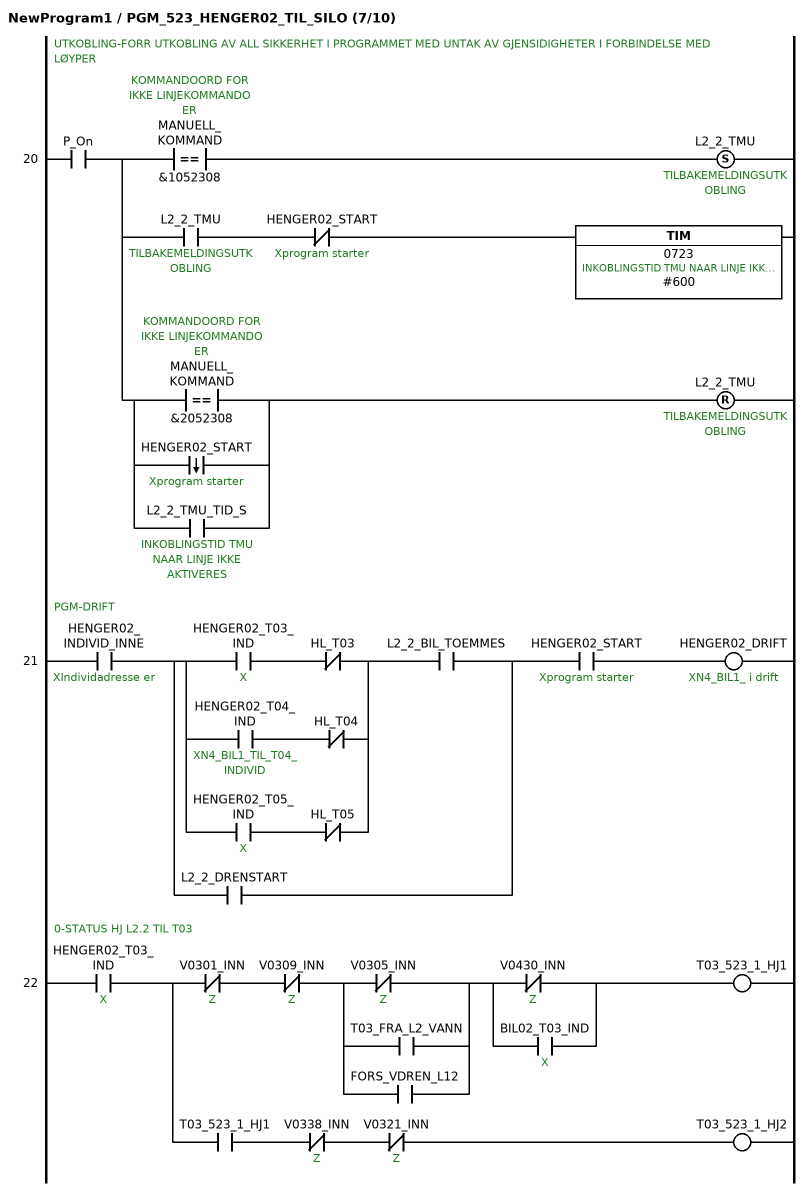
; [picture p648: NewProgram1 / PGM_523_HENGER02_TIL_SILO, rungs 20-22]
; rung 20: UTKOBLING-FORR UTKOBLING AV ALL SIKKERHET I PROGRAMMET MED UNTAK AV GJENSIDIGHETER I FORBINDELSE MED LØYPER
LD P_On
OUT TR0
AND=L(301) MANUELL_KOMMAND &1052308  ; KOMMANDOORD FOR IKKE LINJEKOMMANDOER
SET L2_2_TMU  ; TILBAKEMELDINGSUTKOBLING
LD TR0
AND L2_2_TMU  ; TILBAKEMELDINGSUTKOBLING
ANDNOT HENGER02_START  ; Xprogram starter
TIM 0723 #600  ; INKOBLINGSTID TMU NAAR LINJE IKKE AKTIVERES
LD TR0
LD=L(301) MANUELL_KOMMAND &2052308  ; KOMMANDOORD FOR IKKE LINJEKOMMANDOER
%OR HENGER02_START  ; Xprogram starter
OR L2_2_TMU_TID_S  ; INKOBLINGSTID TMU NAAR LINJE IKKE AKTIVERES
ANDLD
RSET L2_2_TMU  ; TILBAKEMELDINGSUTKOBLING
; rung 21: PGM-DRIFT
LD HENGER02_INDIVID_INNE  ; XIndividadresse er
LD HENGER02_T03_IND  ; X
ANDNOT HL_T03
LD HENGER02_T04_IND  ; XN4_BIL1_TIL_T04_INDIVID
ANDNOT HL_T04
ORLD
LD HENGER02_T05_IND  ; X
ANDNOT HL_T05
ORLD
AND L2_2_BIL_TOEMMES
OR L2_2_DRENSTART
ANDLD
AND HENGER02_START  ; Xprogram starter
OUT HENGER02_DRIFT  ; XN4_BIL1_ i drift
; rung 22: 0-STATUS HJ L2.2 TIL T03
LD HENGER02_T03_IND  ; X
OUT TR0
ANDNOT V0301_INN  ; Z
ANDNOT V0309_INN  ; Z
LDNOT V0305_INN  ; Z
OR T03_FRA_L2_VANN
OR FORS_VDREN_L12
ANDLD
LDNOT V0430_INN  ; Z
OR BIL02_T03_IND  ; X
ANDLD
OUT T03_523_1_HJ1
LD TR0
AND T03_523_1_HJ1
ANDNOT V0338_INN  ; Z
ANDNOT V0321_INN  ; Z
OUT T03_523_1_HJ2

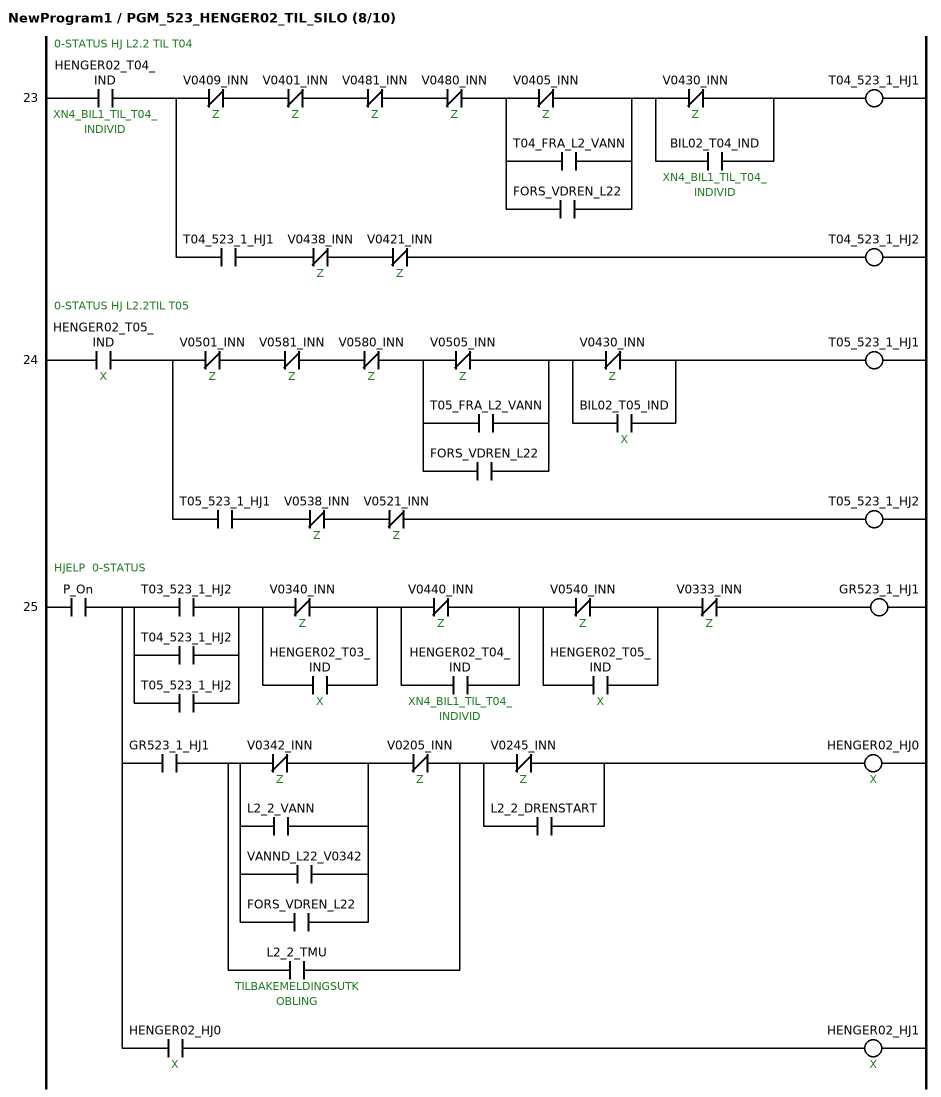
; rung 23: 0-STATUS HJ L2.2 TIL T04
LD HENGER02_T04_IND  ; XN4_BIL1_TIL_T04_INDIVID
OUT TR0
ANDNOT V0409_INN  ; Z
ANDNOT V0401_INN  ; Z
ANDNOT V0481_INN  ; Z
ANDNOT V0480_INN  ; Z
LDNOT V0405_INN  ; Z
OR T04_FRA_L2_VANN
OR FORS_VDREN_L22
ANDLD
LDNOT V0430_INN  ; Z
OR BIL02_T04_IND  ; XN4_BIL1_TIL_T04_INDIVID
ANDLD
OUT T04_523_1_HJ1
LD TR0
AND T04_523_1_HJ1
ANDNOT V0438_INN  ; Z
ANDNOT V0421_INN  ; Z
OUT T04_523_1_HJ2
; rung 24: 0-STATUS HJ L2.2TIL T05
LD HENGER02_T05_IND  ; X
OUT TR0
ANDNOT V0501_INN  ; Z
ANDNOT V0581_INN  ; Z
ANDNOT V0580_INN  ; Z
LDNOT V0505_INN  ; Z
OR T05_FRA_L2_VANN
OR FORS_VDREN_L22
ANDLD
LDNOT V0430_INN  ; Z
OR BIL02_T05_IND  ; X
ANDLD
OUT T05_523_1_HJ1
LD TR0
AND T05_523_1_HJ1
ANDNOT V0538_INN  ; Z
ANDNOT V0521_INN  ; Z
OUT T05_523_1_HJ2
; rung 25: HJELP  0-STATUS
LD P_On
OUT TR0
LD T03_523_1_HJ2
OR T04_523_1_HJ2
OR T05_523_1_HJ2
ANDLD
LDNOT V0340_INN  ; Z
OR HENGER02_T03_IND  ; X
ANDLD
LDNOT V0440_INN  ; Z
OR HENGER02_T04_IND  ; XN4_BIL1_TIL_T04_INDIVID
ANDLD
LDNOT V0540_INN  ; Z
OR HENGER02_T05_IND  ; X
ANDLD
ANDNOT V0333_INN  ; Z
OUT GR523_1_HJ1
LD TR0
AND GR523_1_HJ1
LDNOT V0342_INN  ; Z
OR L2_2_VANN
OR VANND_L22_V0342
OR FORS_VDREN_L22
ANDNOT V0205_INN  ; Z
OR L2_2_TMU  ; TILBAKEMELDINGSUTKOBLING
ANDLD
LDNOT V0245_INN  ; Z
OR L2_2_DRENSTART
ANDLD
OUT HENGER02_HJ0  ; X
LD TR0
AND HENGER02_HJ0  ; X
OUT HENGER02_HJ1  ; X

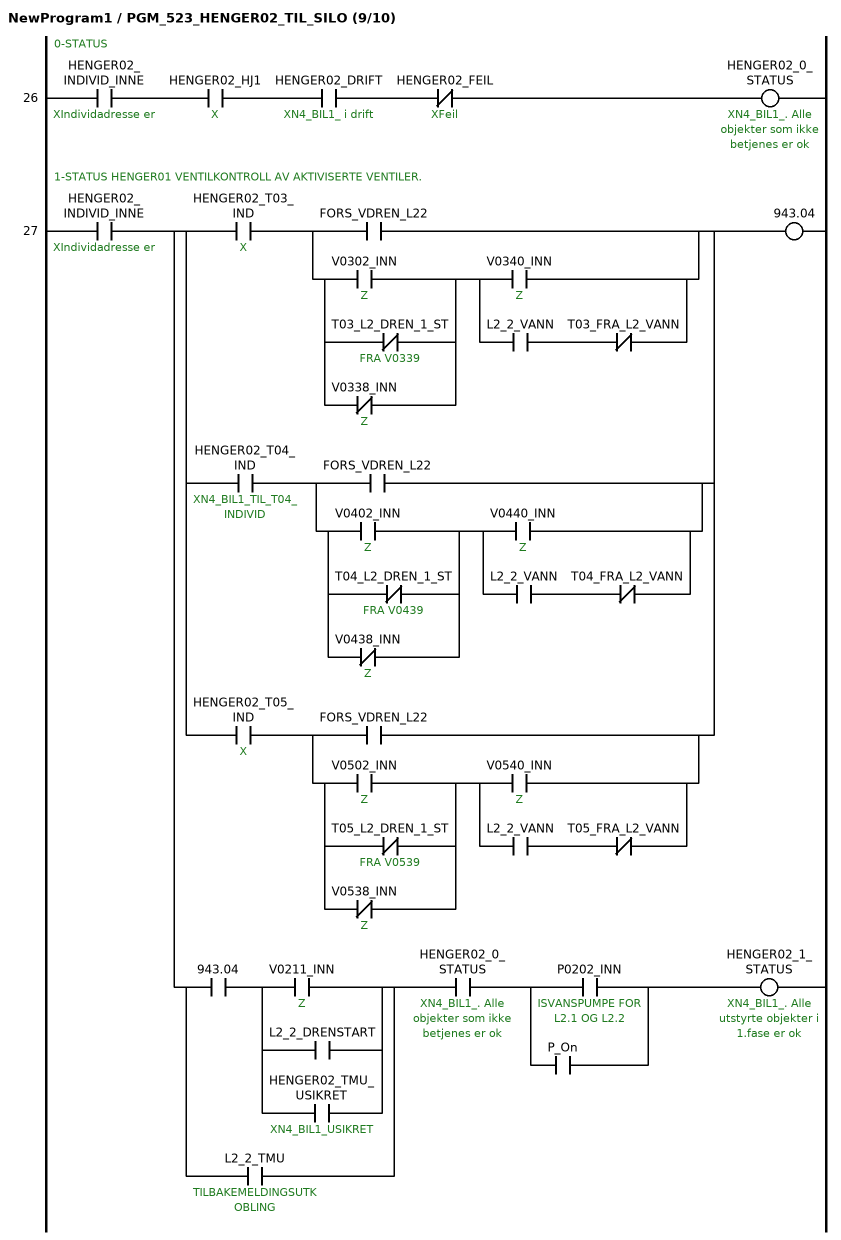
; rung 26: 0-STATUS
LD HENGER02_INDIVID_INNE  ; XIndividadresse er
AND HENGER02_HJ1  ; X
AND HENGER02_DRIFT  ; XN4_BIL1_ i drift
ANDNOT HENGER02_FEIL  ; XFeil
OUT HENGER02_0_STATUS  ; XN4_BIL1_. Alle objekter som ikke betjenes er ok
; rung 27: 1-STATUS HENGER01 VENTILKONTROLL AV AKTIVISERTE VENTILER.
LD HENGER02_INDIVID_INNE  ; XIndividadresse er
OUT TR0
LD HENGER02_T03_IND  ; X
LD FORS_VDREN_L22
LD V0302_INN  ; Z
ORNOT T03_L2_DREN_1_ST  ; FRA V0339
ORNOT V0338_INN  ; Z
LD V0340_INN  ; Z
LD L2_2_VANN
ANDNOT T03_FRA_L2_VANN
ORLD
ANDLD
ORLD
ANDLD
LD HENGER02_T04_IND  ; XN4_BIL1_TIL_T04_INDIVID
LD FORS_VDREN_L22
LD V0402_INN  ; Z
ORNOT T04_L2_DREN_1_ST  ; FRA V0439
ORNOT V0438_INN  ; Z
LD V0440_INN  ; Z
LD L2_2_VANN
ANDNOT T04_FRA_L2_VANN
ORLD
ANDLD
ORLD
ANDLD
ORLD
LD HENGER02_T05_IND  ; X
LD FORS_VDREN_L22
LD V0502_INN  ; Z
ORNOT T05_L2_DREN_1_ST  ; FRA V0539
ORNOT V0538_INN  ; Z
LD V0540_INN  ; Z
LD L2_2_VANN
ANDNOT T05_FRA_L2_VANN
ORLD
ANDLD
ORLD
ANDLD
ORLD
ANDLD
OUT 943.04
LD TR0
LD 943.04
LD V0211_INN  ; Z
OR L2_2_DRENSTART
OR HENGER02_TMU_USIKRET  ; XN4_BIL1_USIKRET
ANDLD
OR L2_2_TMU  ; TILBAKEMELDINGSUTKOBLING
ANDLD
AND HENGER02_0_STATUS  ; XN4_BIL1_. Alle objekter som ikke betjenes er ok
LD P0202_INN  ; ISVANSPUMPE FOR L2.1 OG L2.2
OR P_On
ANDLD
OUT HENGER02_1_STATUS  ; XN4_BIL1_. Alle utstyrte objekter i 1.fase er ok

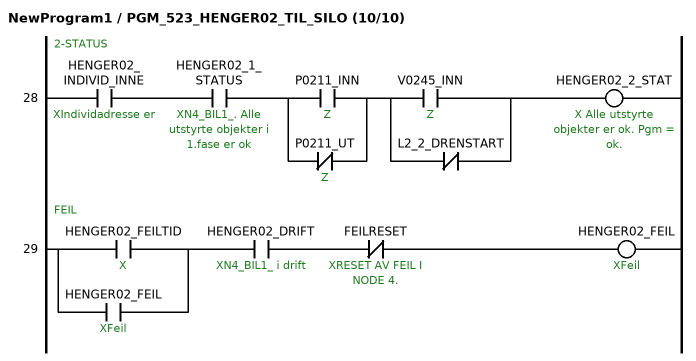
; rung 28: 2-STATUS
LD HENGER02_INDIVID_INNE  ; XIndividadresse er
AND HENGER02_1_STATUS  ; XN4_BIL1_. Alle utstyrte objekter i 1.fase er ok
LD P0211_INN  ; Z
ORNOT P0211_UT  ; Z
ANDLD
LD V0245_INN  ; Z
ORNOT L2_2_DRENSTART
ANDLD
OUT HENGER02_2_STAT  ; X Alle utstyrte objekter er ok. Pgm = ok.
; rung 29: FEIL
LD HENGER02_FEILTID  ; X
OR HENGER02_FEIL  ; XFeil
AND HENGER02_DRIFT  ; XN4_BIL1_ i drift
ANDNOT FEILRESET  ; XRESET AV FEIL I NODE 4.
OUT HENGER02_FEIL  ; XFeil

### Section V0214_P0211

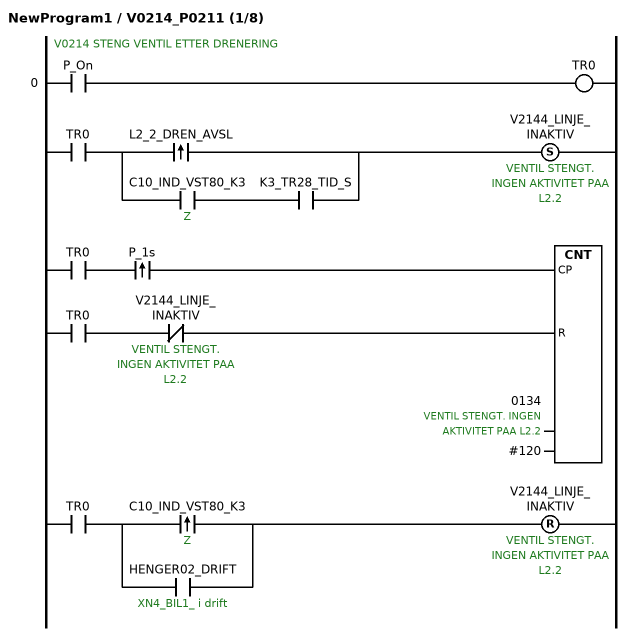
; rung 0: V0214 STENG VENTIL ETTER DRENERING
LD P_On
OUT TR0
@LD L2_2_DREN_AVSL
LD C10_IND_VST80_K3  ; Z
AND K3_TR28_TID_S
ORLD
ANDLD
SET V2144_LINJE_INAKTIV  ; VENTIL STENGT. INGEN AKTIVITET PAA L2.2
LD TR0
@AND P_1s
LD TR0
ANDNOT V2144_LINJE_INAKTIV  ; VENTIL STENGT. INGEN AKTIVITET PAA L2.2
CNT 0134 #120  ; VENTIL STENGT. INGEN AKTIVITET PAA L2.2
LD TR0
@LD C10_IND_VST80_K3  ; Z
OR HENGER02_DRIFT  ; XN4_BIL1_ i drift
ANDLD
RSET V2144_LINJE_INAKTIV  ; VENTIL STENGT. INGEN AKTIVITET PAA L2.2

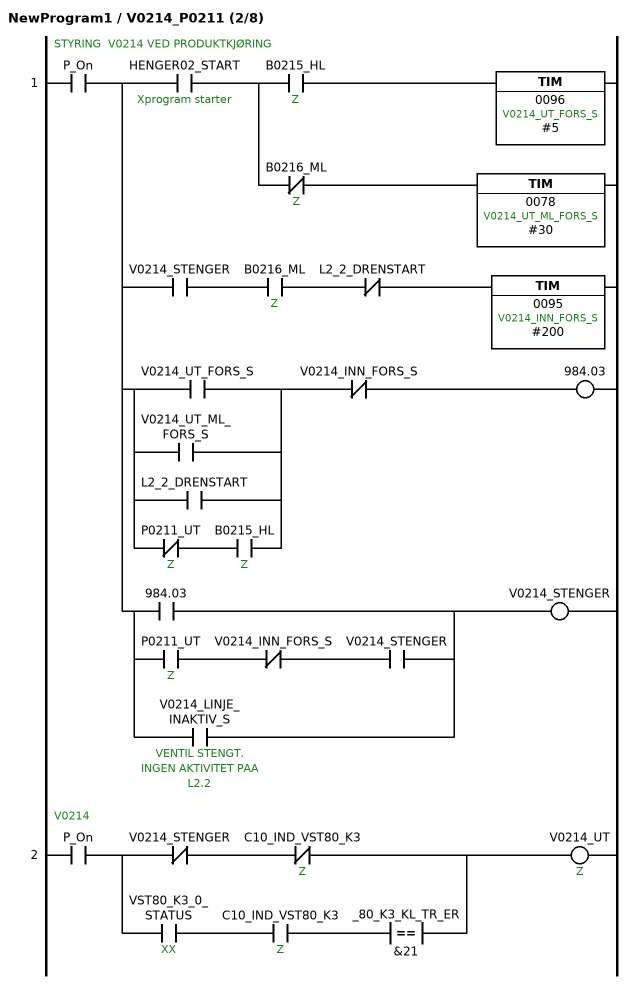
; rung 1: STYRING  V0214 VED PRODUKTKJØRING
LD P_On
OUT TR0
AND HENGER02_START  ; Xprogram starter
OUT TR1
AND B0215_HL  ; Z
TIM 0096 #5  ; V0214_UT_FORS_S
LD TR1
ANDNOT B0216_ML  ; Z
TIM 0078 #30  ; V0214_UT_ML_FORS_S
LD TR0
AND V0214_STENGER
AND B0216_ML  ; Z
ANDNOT L2_2_DRENSTART
TIM 0095 #200  ; V0214_INN_FORS_S
LD TR0
LD V0214_UT_FORS_S
OR V0214_UT_ML_FORS_S
OR L2_2_DRENSTART
LDNOT P0211_UT  ; Z
AND B0215_HL  ; Z
ORLD
ANDLD
ANDNOT V0214_INN_FORS_S
OUT 984.03
LD TR0
LD 984.03
LD P0211_UT  ; Z
ANDNOT V0214_INN_FORS_S
AND V0214_STENGER
ORLD
OR V0214_LINJE_INAKTIV_S  ; VENTIL STENGT. INGEN AKTIVITET PAA L2.2
ANDLD
OUT V0214_STENGER
; rung 2: V0214
LD P_On
LDNOT V0214_STENGER
ANDNOT C10_IND_VST80_K3  ; Z
LD VST80_K3_0_STATUS  ; XX
AND C10_IND_VST80_K3  ; Z
AND=(300) _80_K3_KL_TR_ER &21
ORLD
ANDLD
OUT V0214_UT  ; Z

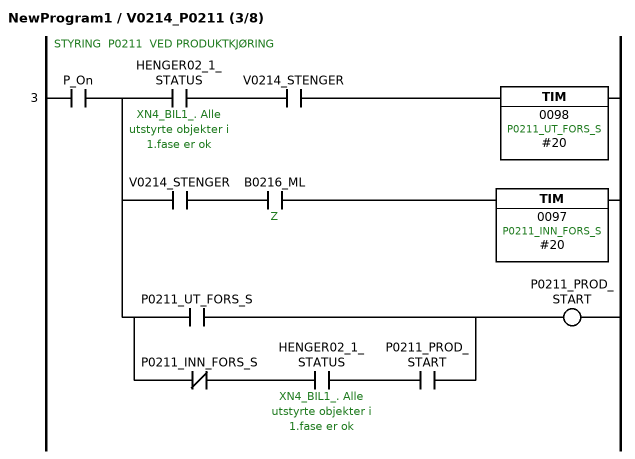
; rung 3: STYRING  P0211  VED PRODUKTKJØRING
LD P_On
OUT TR0
AND HENGER02_1_STATUS  ; XN4_BIL1_. Alle utstyrte objekter i 1.fase er ok
AND V0214_STENGER
TIM 0098 #20  ; P0211_UT_FORS_S
LD TR0
AND V0214_STENGER
AND B0216_ML  ; Z
TIM 0097 #20  ; P0211_INN_FORS_S
LD TR0
LD P0211_UT_FORS_S
LDNOT P0211_INN_FORS_S
AND HENGER02_1_STATUS  ; XN4_BIL1_. Alle utstyrte objekter i 1.fase er ok
AND P0211_PROD_START
ORLD
ANDLD
OUT P0211_PROD_START

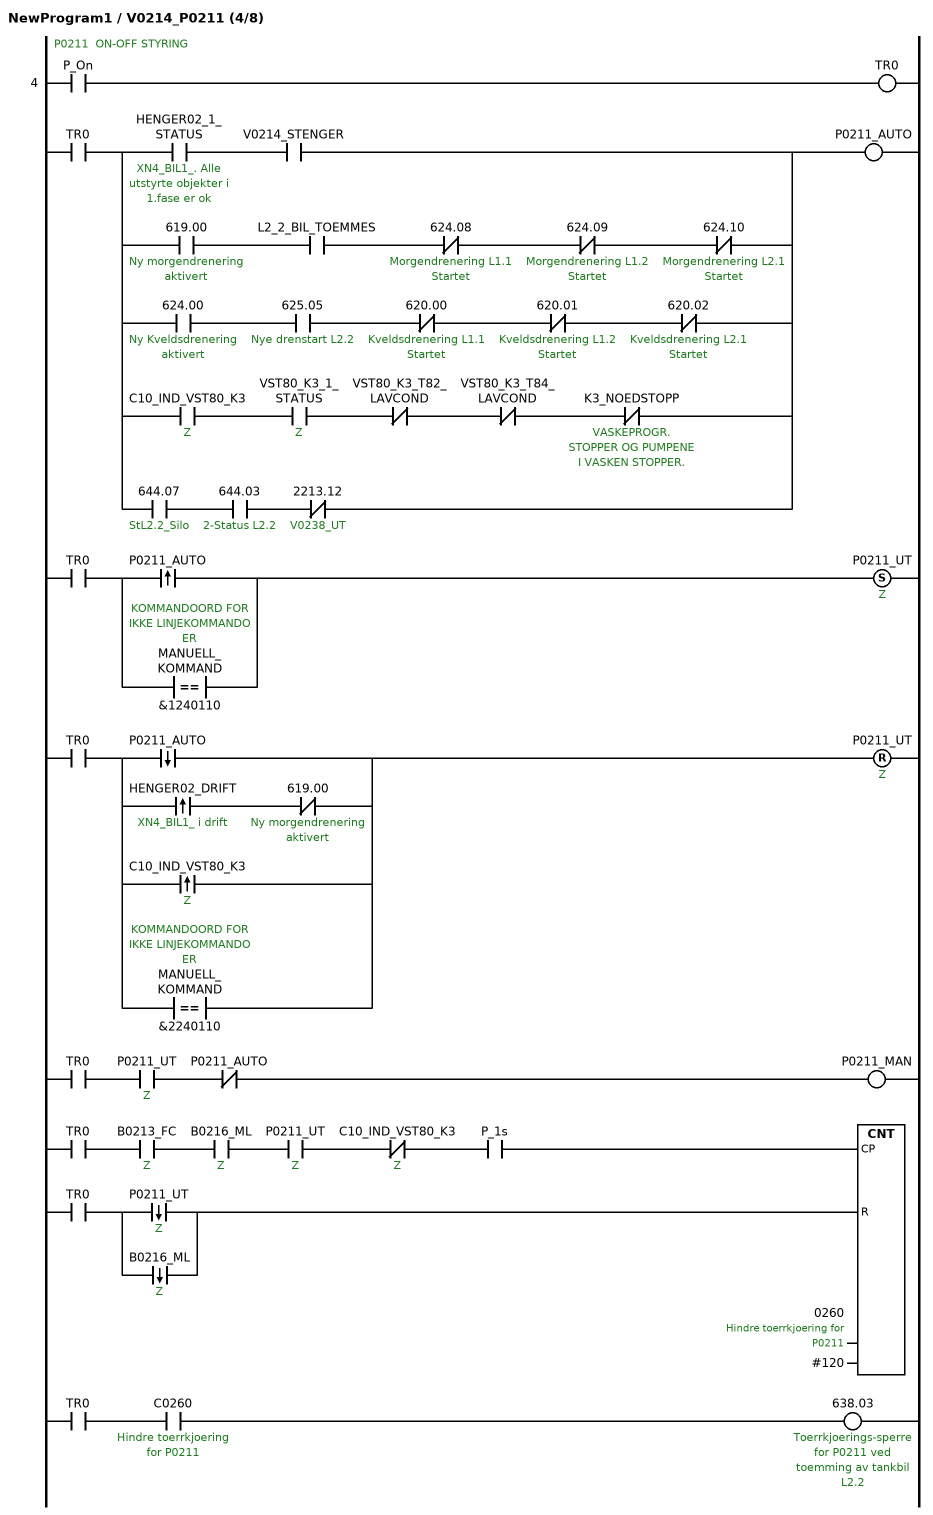
; rung 4: P0211  ON-OFF STYRING
LD P_On
OUT TR0
LD HENGER02_1_STATUS  ; XN4_BIL1_. Alle utstyrte objekter i 1.fase er ok
AND V0214_STENGER
LD 619.00  ; Ny morgendrenering aktivert
AND L2_2_BIL_TOEMMES
ANDNOT 624.08  ; Morgendrenering L1.1 Startet
ANDNOT 624.09  ; Morgendrenering L1.2 Startet
ANDNOT 624.10  ; Morgendrenering L2.1 Startet
ORLD
LD 624.00  ; Ny Kveldsdrenering aktivert
AND 625.05  ; Nye drenstart L2.2
ANDNOT 620.00  ; Kveldsdrenering L1.1 Startet
ANDNOT 620.01  ; Kveldsdrenering L1.2 Startet
ANDNOT 620.02  ; Kveldsdrenering L2.1 Startet
ORLD
LD C10_IND_VST80_K3  ; Z
AND VST80_K3_1_STATUS  ; Z
ANDNOT VST80_K3_T82_LAVCOND
ANDNOT VST80_K3_T84_LAVCOND
ANDNOT K3_NOEDSTOPP  ; VASKEPROGR. STOPPER OG PUMPENE I VASKEN STOPPER.
ORLD
LD 644.07  ; StL2.2_Silo
AND 644.03  ; 2-Status L2.2
ANDNOT 2213.12  ; V0238_UT
ORLD
ANDLD
OUT P0211_AUTO
LD TR0
@LD P0211_AUTO
OR=L(301) MANUELL_KOMMAND &1240110  ; KOMMANDOORD FOR IKKE LINJEKOMMANDOER
ANDLD
SET P0211_UT  ; Z
LD TR0
%LD P0211_AUTO
@LD HENGER02_DRIFT  ; XN4_BIL1_ i drift
ANDNOT 619.00  ; Ny morgendrenering aktivert
ORLD
@OR C10_IND_VST80_K3  ; Z
OR=L(301) MANUELL_KOMMAND &2240110  ; KOMMANDOORD FOR IKKE LINJEKOMMANDOER
ANDLD
RSET P0211_UT  ; Z
LD TR0
AND P0211_UT  ; Z
ANDNOT P0211_AUTO
OUT P0211_MAN
LD TR0
AND B0213_FC  ; Z
AND B0216_ML  ; Z
AND P0211_UT  ; Z
ANDNOT C10_IND_VST80_K3  ; Z
AND P_1s
LD TR0
%LD P0211_UT  ; Z
%OR B0216_ML  ; Z
ANDLD
CNT 0260 #120  ; Hindre toerrkjoering for P0211
LD TR0
AND C0260  ; Hindre toerrkjoering for P0211
OUT 638.03  ; Toerrkjoerings-sperre for P0211 ved toemming av tankbil L2.2

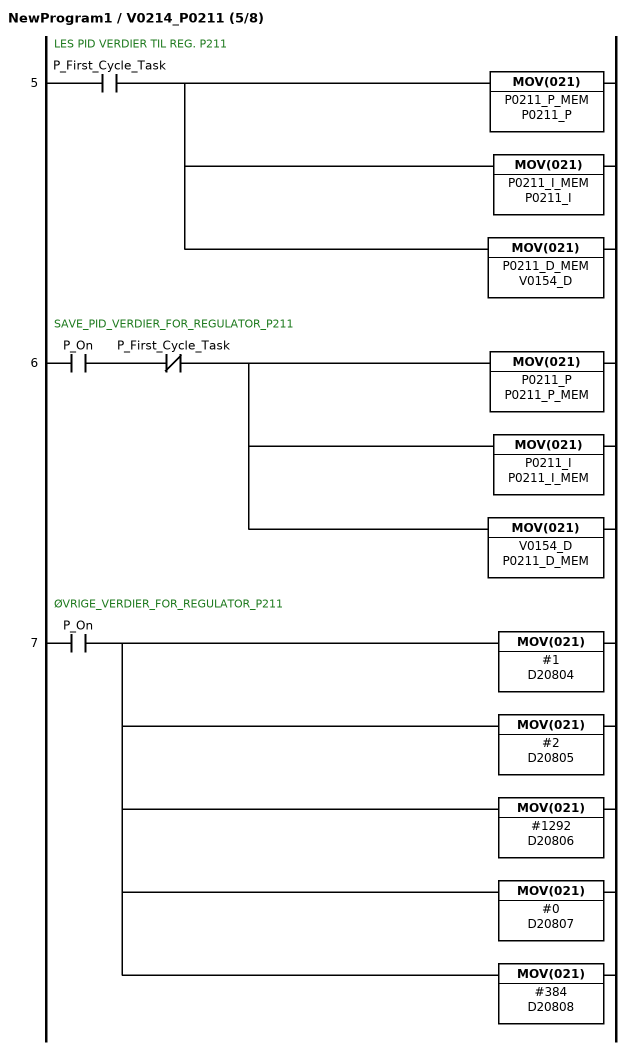
; rung 5: LES PID VERDIER TIL REG. P211
LD P_First_Cycle_Task
MOV(021) P0211_P_MEM P0211_P
MOV(021) P0211_I_MEM P0211_I
MOV(021) P0211_D_MEM V0154_D
; rung 6: SAVE_PID_VERDIER_FOR_REGULATOR_P211
LD P_On
ANDNOT P_First_Cycle_Task
MOV(021) P0211_P P0211_P_MEM
MOV(021) P0211_I P0211_I_MEM
MOV(021) V0154_D P0211_D_MEM
; rung 7: ØVRIGE_VERDIER_FOR_REGULATOR_P211
LD P_On
MOV(021) #1 D20804
MOV(021) #2 D20805
MOV(021) #1292 D20806
MOV(021) #0 D20807
MOV(021) #384 D20808

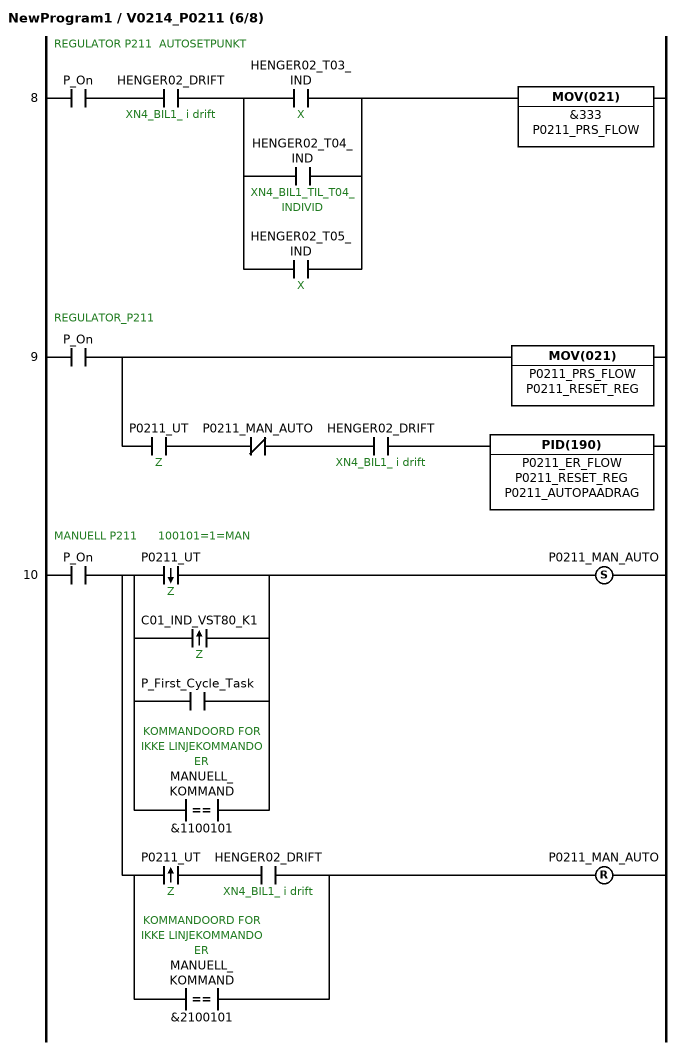
; rung 8: REGULATOR P211  AUTOSETPUNKT
LD P_On
AND HENGER02_DRIFT  ; XN4_BIL1_ i drift
LD HENGER02_T03_IND  ; X
OR HENGER02_T04_IND  ; XN4_BIL1_TIL_T04_INDIVID
OR HENGER02_T05_IND  ; X
ANDLD
MOV(021) &333 P0211_PRS_FLOW
; rung 9: REGULATOR_P211
LD P_On
MOV(021) P0211_PRS_FLOW P0211_RESET_REG
AND P0211_UT  ; Z
ANDNOT P0211_MAN_AUTO
AND HENGER02_DRIFT  ; XN4_BIL1_ i drift
PID(190) P0211_ER_FLOW P0211_RESET_REG P0211_AUTOPAADRAG
; rung 10: MANUELL P211      100101=1=MAN
LD P_On
OUT TR0
%LD P0211_UT  ; Z
@OR C01_IND_VST80_K1  ; Z
OR P_First_Cycle_Task
OR=L(301) MANUELL_KOMMAND &1100101  ; KOMMANDOORD FOR IKKE LINJEKOMMANDOER
ANDLD
SET P0211_MAN_AUTO
LD TR0
@LD P0211_UT  ; Z
AND HENGER02_DRIFT  ; XN4_BIL1_ i drift
OR=L(301) MANUELL_KOMMAND &2100101  ; KOMMANDOORD FOR IKKE LINJEKOMMANDOER
ANDLD
RSET P0211_MAN_AUTO

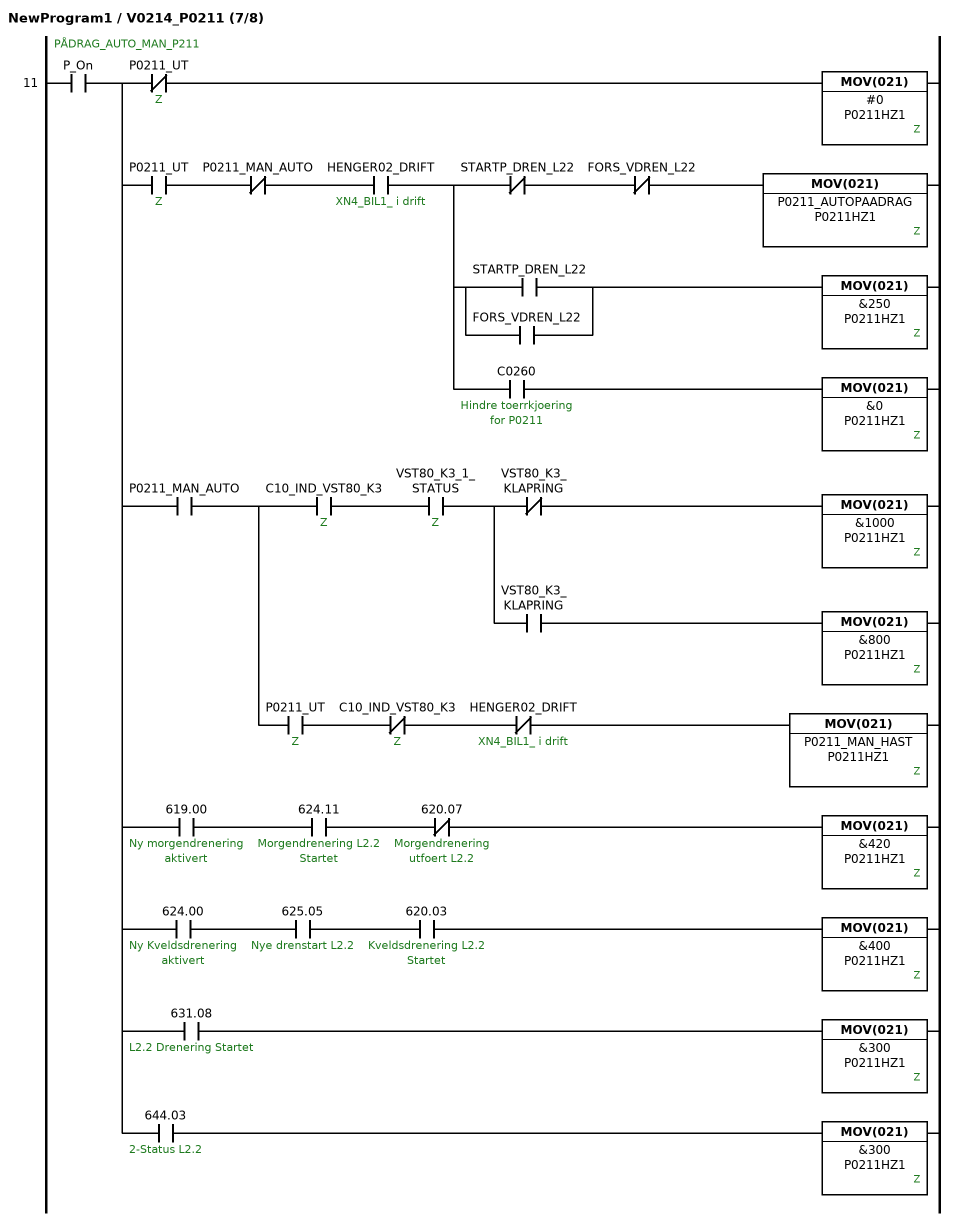
; rung 11: PÅDRAG_AUTO_MAN_P211
LD P_On
OUT TR0
ANDNOT P0211_UT  ; Z
MOV(021) #0 P0211HZ1  ; Z
LD TR0
AND P0211_UT  ; Z
ANDNOT P0211_MAN_AUTO
AND HENGER02_DRIFT  ; XN4_BIL1_ i drift
OUT TR1
ANDNOT STARTP_DREN_L22
ANDNOT FORS_VDREN_L22
MOV(021) P0211_AUTOPAADRAG P0211HZ1  ; Z
LD TR1
LD STARTP_DREN_L22
OR FORS_VDREN_L22
ANDLD
MOV(021) &250 P0211HZ1  ; Z
LD TR1
AND C0260  ; Hindre toerrkjoering for P0211
MOV(021) &0 P0211HZ1  ; Z
LD TR0
AND P0211_MAN_AUTO
OUT TR1
AND C10_IND_VST80_K3  ; Z
AND VST80_K3_1_STATUS  ; Z
OUT TR2
ANDNOT VST80_K3_KLAPRING
MOV(021) &1000 P0211HZ1  ; Z
LD TR2
AND VST80_K3_KLAPRING
MOV(021) &800 P0211HZ1  ; Z
LD TR1
AND P0211_UT  ; Z
ANDNOT C10_IND_VST80_K3  ; Z
ANDNOT HENGER02_DRIFT  ; XN4_BIL1_ i drift
MOV(021) P0211_MAN_HAST P0211HZ1  ; Z
LD TR0
AND 619.00  ; Ny morgendrenering aktivert
AND 624.11  ; Morgendrenering L2.2 Startet
ANDNOT 620.07  ; Morgendrenering utfoert L2.2
MOV(021) &420 P0211HZ1  ; Z
LD TR0
AND 624.00  ; Ny Kveldsdrenering aktivert
AND 625.05  ; Nye drenstart L2.2
AND 620.03  ; Kveldsdrenering L2.2 Startet
MOV(021) &400 P0211HZ1  ; Z
LD TR0
AND 631.08  ; L2.2 Drenering Startet
MOV(021) &300 P0211HZ1  ; Z
LD TR0
AND 644.03  ; 2-Status L2.2
MOV(021) &300 P0211HZ1  ; Z

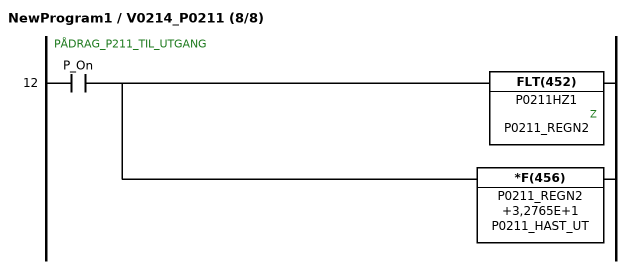
; rung 12: PÅDRAG_P211_TIL_UTGANG
LD P_On
FLT(452) P0211HZ1 P0211_REGN2  ; Z
*F(456) P0211_REGN2 +3,2765E+1 P0211_HAST_UT

### Section V251_V0254_ISV

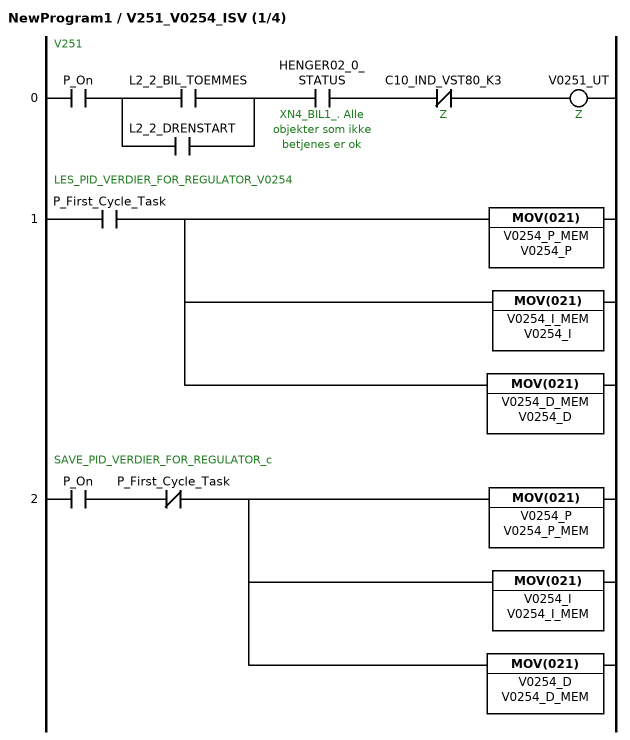
; rung 0: V251
LD P_On
LD L2_2_BIL_TOEMMES
OR L2_2_DRENSTART
ANDLD
AND HENGER02_0_STATUS  ; XN4_BIL1_. Alle objekter som ikke betjenes er ok
ANDNOT C10_IND_VST80_K3  ; Z
OUT V0251_UT  ; Z
; rung 1: LES_PID_VERDIER_FOR_REGULATOR_V0254
LD P_First_Cycle_Task
MOV(021) V0254_P_MEM V0254_P
MOV(021) V0254_I_MEM V0254_I
MOV(021) V0254_D_MEM V0254_D
; rung 2: SAVE_PID_VERDIER_FOR_REGULATOR_c
LD P_On
ANDNOT P_First_Cycle_Task
MOV(021) V0254_P V0254_P_MEM
MOV(021) V0254_I V0254_I_MEM
MOV(021) V0254_D V0254_D_MEM

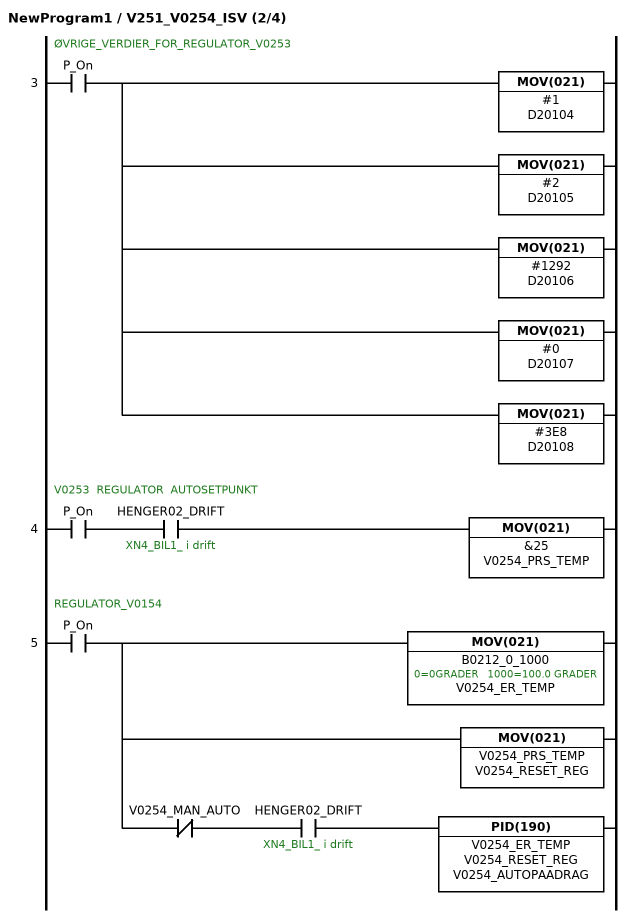
; rung 3: ØVRIGE_VERDIER_FOR_REGULATOR_V0253
LD P_On
MOV(021) #1 D20104
MOV(021) #2 D20105
MOV(021) #1292 D20106
MOV(021) #0 D20107
MOV(021) #3E8 D20108
; rung 4: V0253  REGULATOR  AUTOSETPUNKT
LD P_On
AND HENGER02_DRIFT  ; XN4_BIL1_ i drift
MOV(021) &25 V0254_PRS_TEMP
; rung 5: REGULATOR_V0154
LD P_On
MOV(021) B0212_0_1000 V0254_ER_TEMP  ; 0=0GRADER   1000=100.0 GRADER
MOV(021) V0254_PRS_TEMP V0254_RESET_REG
ANDNOT V0254_MAN_AUTO
AND HENGER02_DRIFT  ; XN4_BIL1_ i drift
PID(190) V0254_ER_TEMP V0254_RESET_REG V0254_AUTOPAADRAG

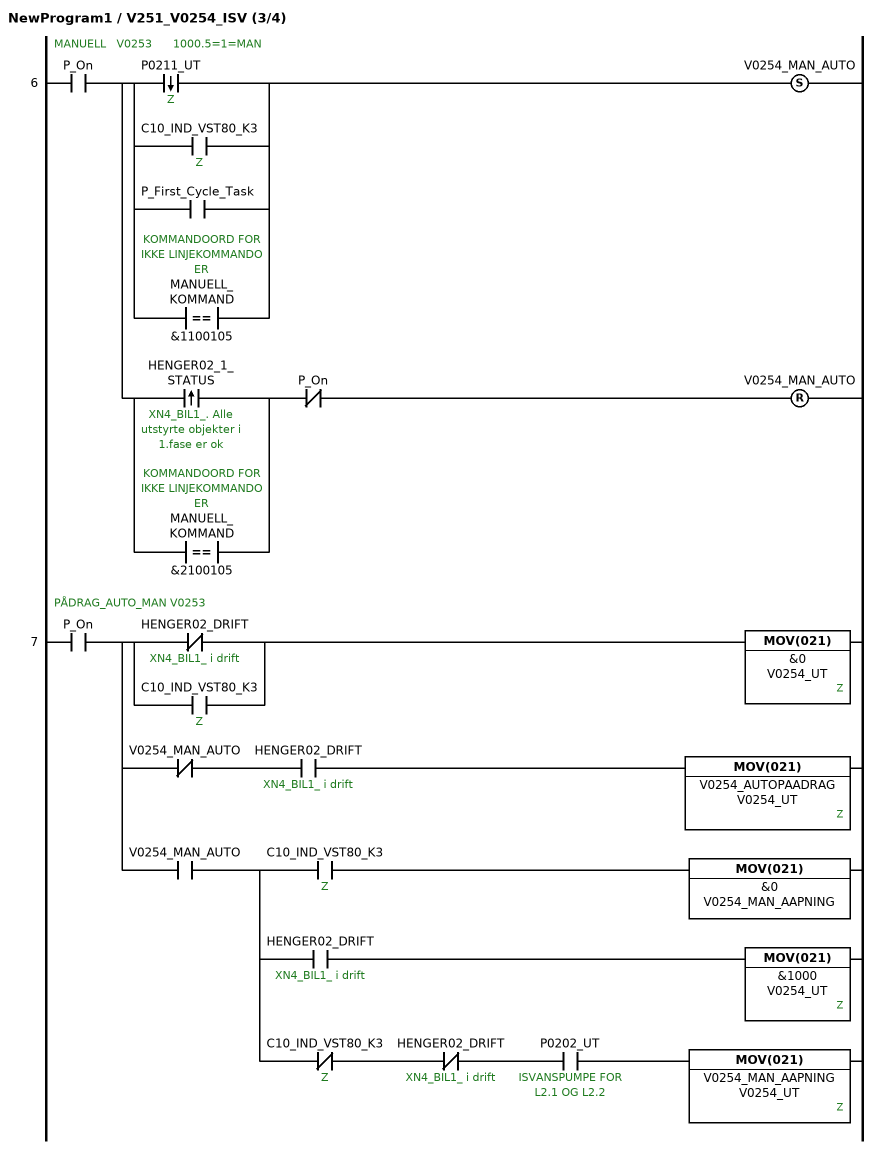
; rung 6: MANUELL   V0253      1000.5=1=MAN
LD P_On
OUT TR0
%LD P0211_UT  ; Z
OR C10_IND_VST80_K3  ; Z
OR P_First_Cycle_Task
OR=L(301) MANUELL_KOMMAND &1100105  ; KOMMANDOORD FOR IKKE LINJEKOMMANDOER
ANDLD
SET V0254_MAN_AUTO
LD TR0
@LD HENGER02_1_STATUS  ; XN4_BIL1_. Alle utstyrte objekter i 1.fase er ok
OR=L(301) MANUELL_KOMMAND &2100105  ; KOMMANDOORD FOR IKKE LINJEKOMMANDOER
ANDLD
ANDNOT P_On
RSET V0254_MAN_AUTO
; rung 7: PÅDRAG_AUTO_MAN V0253
LD P_On
OUT TR0
LDNOT HENGER02_DRIFT  ; XN4_BIL1_ i drift
OR C10_IND_VST80_K3  ; Z
ANDLD
MOV(021) &0 V0254_UT  ; Z
LD TR0
ANDNOT V0254_MAN_AUTO
AND HENGER02_DRIFT  ; XN4_BIL1_ i drift
MOV(021) V0254_AUTOPAADRAG V0254_UT  ; Z
LD TR0
AND V0254_MAN_AUTO
OUT TR0
AND C10_IND_VST80_K3  ; Z
MOV(021) &0 V0254_MAN_AAPNING
LD TR0
AND HENGER02_DRIFT  ; XN4_BIL1_ i drift
MOV(021) &1000 V0254_UT  ; Z
LD TR0
ANDNOT C10_IND_VST80_K3  ; Z
ANDNOT HENGER02_DRIFT  ; XN4_BIL1_ i drift
AND P0202_UT  ; ISVANSPUMPE FOR L2.1 OG L2.2
MOV(021) V0254_MAN_AAPNING V0254_UT  ; Z

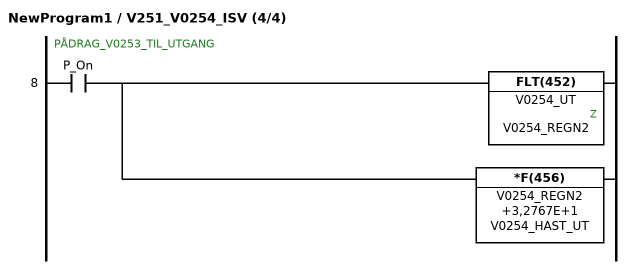
; rung 8: PÅDRAG_V0253_TIL_UTGANG
LD P_On
FLT(452) V0254_UT V0254_REGN2  ; Z
*F(456) V0254_REGN2 +3,2767E+1 V0254_HAST_UT

### Section PGM524_SILO_TIL_L3

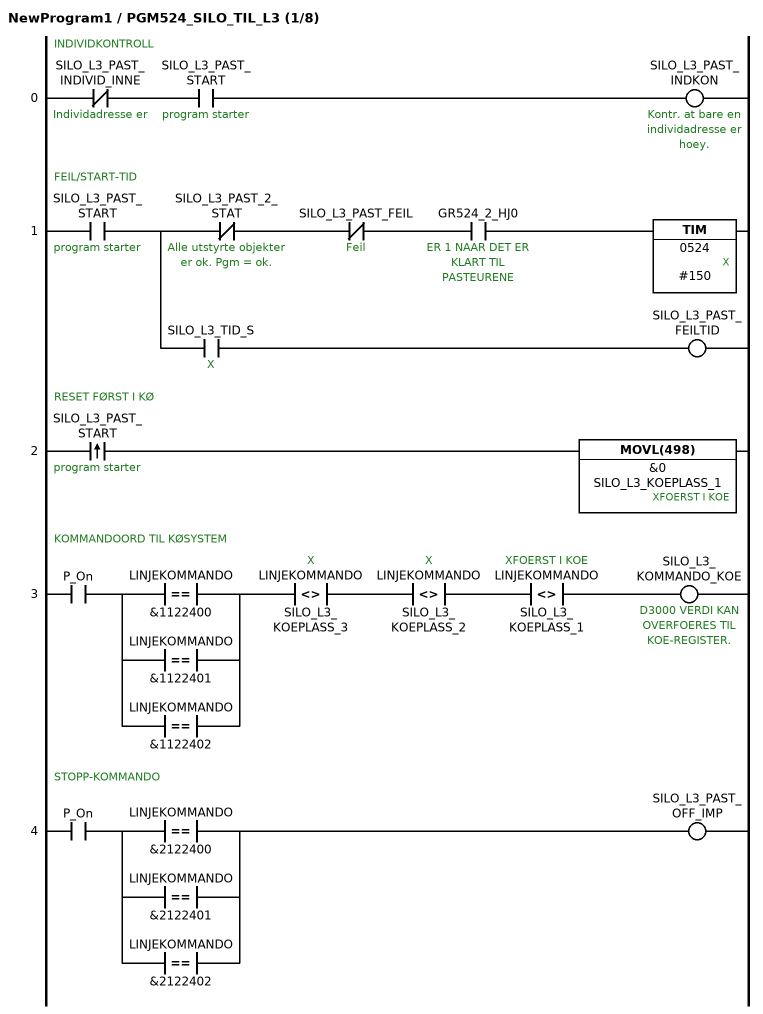
; rung 0: INDIVIDKONTROLL
LDNOT SILO_L3_PAST_INDIVID_INNE  ; Individadresse er
AND SILO_L3_PAST_START  ; program starter
OUT SILO_L3_PAST_INDKON  ; Kontr. at bare en individadresse er hoey.
; rung 1: FEIL/START-TID
LD SILO_L3_PAST_START  ; program starter
OUT TR0
ANDNOT SILO_L3_PAST_2_STAT  ; Alle utstyrte objekter er ok. Pgm = ok.
ANDNOT SILO_L3_PAST_FEIL  ; Feil
AND GR524_2_HJ0  ; ER 1 NAAR DET ER KLART TIL PASTEURENE
TIM 0524 #150  ; X
LD TR0
AND SILO_L3_TID_S  ; X
OUT SILO_L3_PAST_FEILTID
; rung 2: RESET FØRST I KØ
@LD SILO_L3_PAST_START  ; program starter
MOVL(498) &0 SILO_L3_KOEPLASS_1  ; XFOERST I KOE
; rung 3: KOMMANDOORD TIL KØSYSTEM
LD P_On
LD=L(301) LINJEKOMMANDO &1122400
OR=L(301) LINJEKOMMANDO &1122401
OR=L(301) LINJEKOMMANDO &1122402
ANDLD
AND<>L(306) LINJEKOMMANDO SILO_L3_KOEPLASS_3  ; X
AND<>L(306) LINJEKOMMANDO SILO_L3_KOEPLASS_2  ; X
AND<>L(306) LINJEKOMMANDO SILO_L3_KOEPLASS_1  ; XFOERST I KOE
OUT SILO_L3_KOMMANDO_KOE  ; D3000 VERDI KAN OVERFOERES TIL KOE-REGISTER.
; rung 4: STOPP-KOMMANDO
LD P_On
LD=L(301) LINJEKOMMANDO &2122400
OR=L(301) LINJEKOMMANDO &2122401
OR=L(301) LINJEKOMMANDO &2122402
ANDLD
OUT SILO_L3_PAST_OFF_IMP

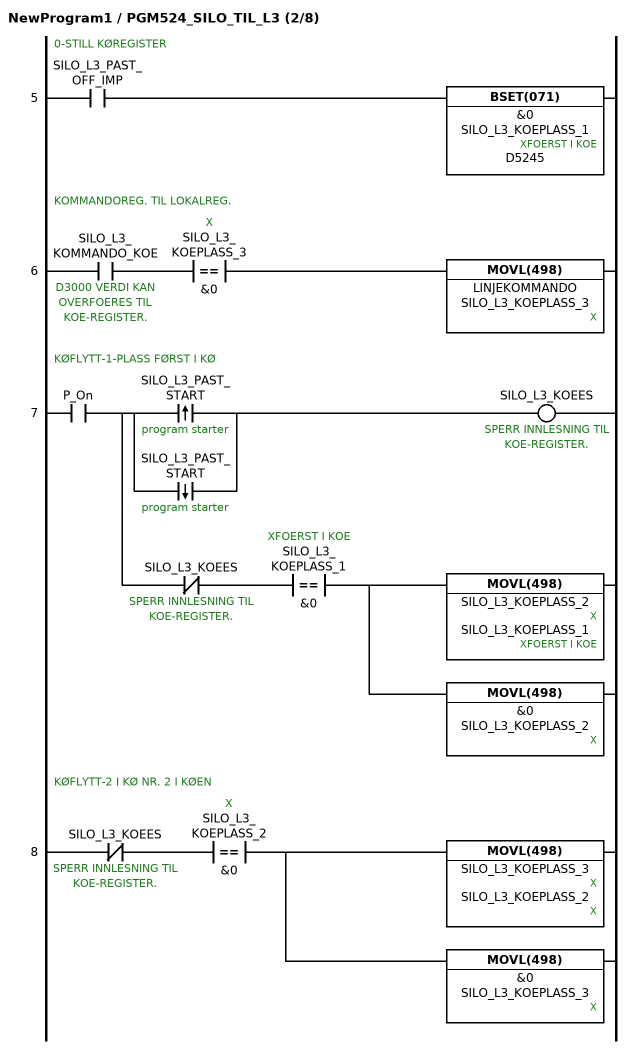
; rung 5: 0-STILL KØREGISTER
LD SILO_L3_PAST_OFF_IMP
BSET(071) &0 SILO_L3_KOEPLASS_1 D5245  ; XFOERST I KOE
; rung 6: KOMMANDOREG. TIL LOKALREG.
LD SILO_L3_KOMMANDO_KOE  ; D3000 VERDI KAN OVERFOERES TIL KOE-REGISTER.
AND=L(301) SILO_L3_KOEPLASS_3 &0  ; X
MOVL(498) LINJEKOMMANDO SILO_L3_KOEPLASS_3  ; X
; rung 7: KØFLYTT-1-PLASS FØRST I KØ
LD P_On
OUT TR0
@LD SILO_L3_PAST_START  ; program starter
%OR SILO_L3_PAST_START  ; program starter
ANDLD
OUT SILO_L3_KOEES  ; SPERR INNLESNING TIL KOE-REGISTER.
LD TR0
ANDNOT SILO_L3_KOEES  ; SPERR INNLESNING TIL KOE-REGISTER.
AND=L(301) SILO_L3_KOEPLASS_1 &0  ; XFOERST I KOE
MOVL(498) SILO_L3_KOEPLASS_2 SILO_L3_KOEPLASS_1  ; X, XFOERST I KOE
MOVL(498) &0 SILO_L3_KOEPLASS_2  ; X
; rung 8: KØFLYTT-2 I KØ NR. 2 I KØEN
LDNOT SILO_L3_KOEES  ; SPERR INNLESNING TIL KOE-REGISTER.
AND=L(301) SILO_L3_KOEPLASS_2 &0  ; X
MOVL(498) SILO_L3_KOEPLASS_3 SILO_L3_KOEPLASS_2  ; X
MOVL(498) &0 SILO_L3_KOEPLASS_3  ; X

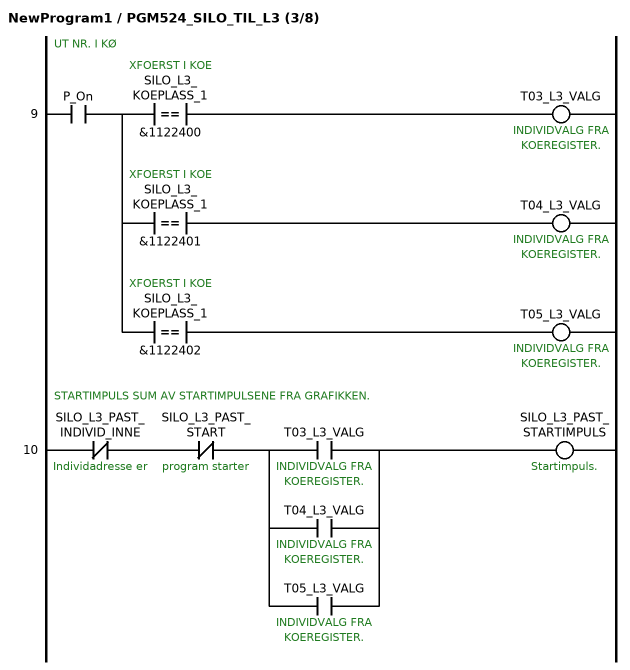
; rung 9: UT NR. I KØ
LD P_On
OUT TR0
AND=L(301) SILO_L3_KOEPLASS_1 &1122400  ; XFOERST I KOE
OUT T03_L3_VALG  ; INDIVIDVALG FRA KOEREGISTER.
LD TR0
AND=L(301) SILO_L3_KOEPLASS_1 &1122401  ; XFOERST I KOE
OUT T04_L3_VALG  ; INDIVIDVALG FRA KOEREGISTER.
LD TR0
AND=L(301) SILO_L3_KOEPLASS_1 &1122402  ; XFOERST I KOE
OUT T05_L3_VALG  ; INDIVIDVALG FRA KOEREGISTER.
; rung 10: STARTIMPULS SUM AV STARTIMPULSENE FRA GRAFIKKEN.
LDNOT SILO_L3_PAST_INDIVID_INNE  ; Individadresse er
ANDNOT SILO_L3_PAST_START  ; program starter
LD T03_L3_VALG  ; INDIVIDVALG FRA KOEREGISTER.
OR T04_L3_VALG  ; INDIVIDVALG FRA KOEREGISTER.
OR T05_L3_VALG  ; INDIVIDVALG FRA KOEREGISTER.
ANDLD
OUT SILO_L3_PAST_STARTIMPULS  ; Startimpuls.

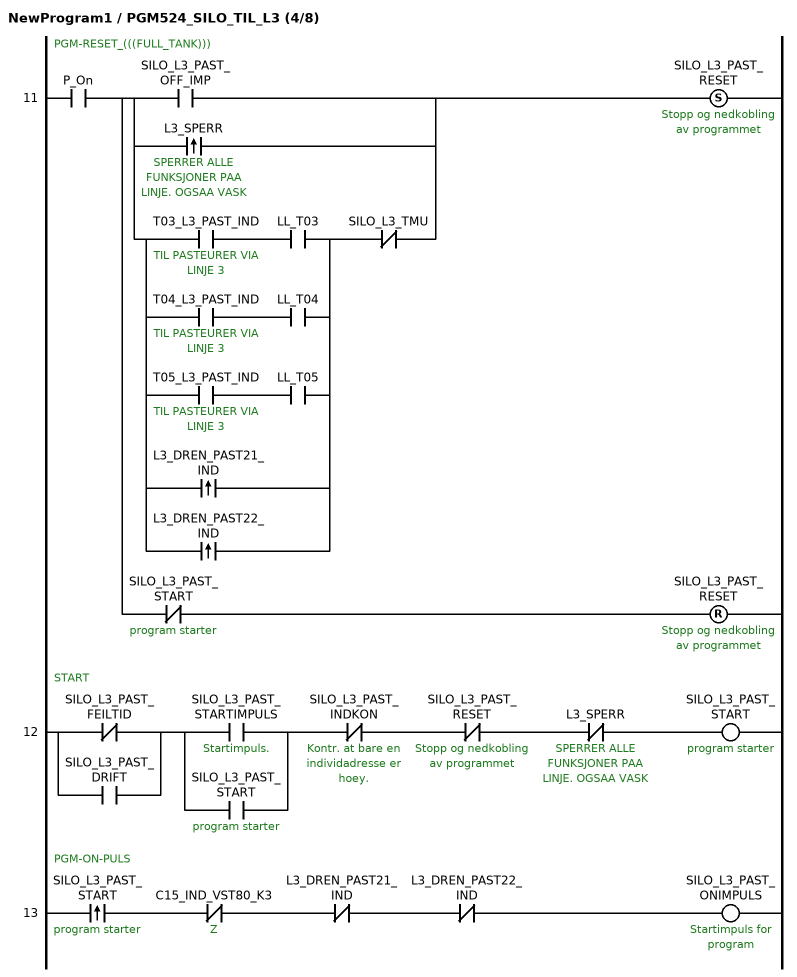
; rung 11: PGM-RESET_(((FULL_TANK)))
LD P_On
OUT TR0
LD SILO_L3_PAST_OFF_IMP
@OR L3_SPERR  ; SPERRER ALLE FUNKSJONER PAA LINJE. OGSAA VASK
LD T03_L3_PAST_IND  ; TIL PASTEURER VIA LINJE 3
AND LL_T03
LD T04_L3_PAST_IND  ; TIL PASTEURER VIA LINJE 3
AND LL_T04
ORLD
LD T05_L3_PAST_IND  ; TIL PASTEURER VIA LINJE 3
AND LL_T05
ORLD
@OR L3_DREN_PAST21_IND
@OR L3_DREN_PAST22_IND
ANDNOT SILO_L3_TMU
ORLD
ANDLD
SET SILO_L3_PAST_RESET  ; Stopp og nedkobling av programmet
LD TR0
ANDNOT SILO_L3_PAST_START  ; program starter
RSET SILO_L3_PAST_RESET  ; Stopp og nedkobling av programmet
; rung 12: START
LDNOT SILO_L3_PAST_FEILTID
OR SILO_L3_PAST_DRIFT
LD SILO_L3_PAST_STARTIMPULS  ; Startimpuls.
OR SILO_L3_PAST_START  ; program starter
ANDLD
ANDNOT SILO_L3_PAST_INDKON  ; Kontr. at bare en individadresse er hoey.
ANDNOT SILO_L3_PAST_RESET  ; Stopp og nedkobling av programmet
ANDNOT L3_SPERR  ; SPERRER ALLE FUNKSJONER PAA LINJE. OGSAA VASK
OUT SILO_L3_PAST_START  ; program starter
; rung 13: PGM-ON-PULS
@LD SILO_L3_PAST_START  ; program starter
ANDNOT C15_IND_VST80_K3  ; Z
ANDNOT L3_DREN_PAST21_IND
ANDNOT L3_DREN_PAST22_IND
OUT SILO_L3_PAST_ONIMPULS  ; Startimpuls for  program

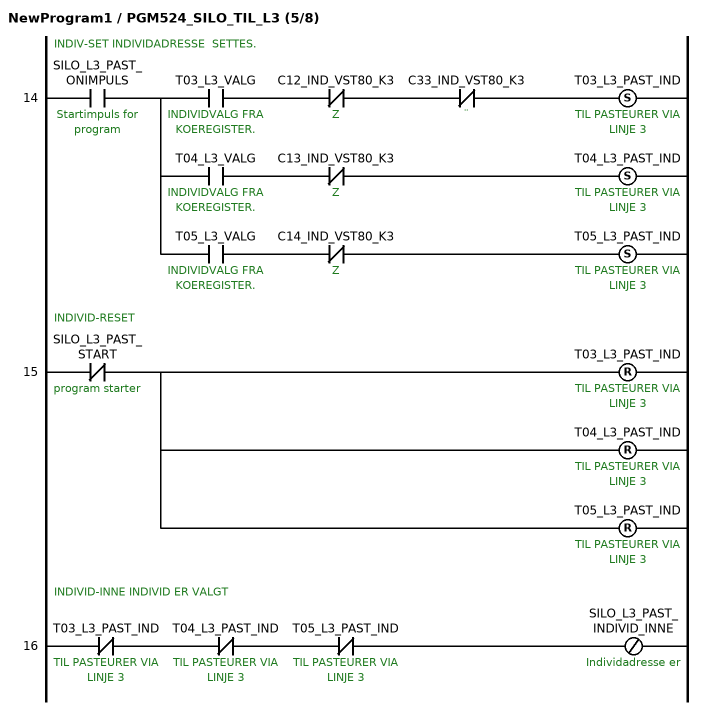
; rung 14: INDIV-SET INDIVIDADRESSE  SETTES.
LD SILO_L3_PAST_ONIMPULS  ; Startimpuls for  program
OUT TR0
AND T03_L3_VALG  ; INDIVIDVALG FRA KOEREGISTER.
ANDNOT C12_IND_VST80_K3  ; Z
ANDNOT C33_IND_VST80_K3  ; ¨
SET T03_L3_PAST_IND  ; TIL PASTEURER VIA LINJE 3
LD TR0
AND T04_L3_VALG  ; INDIVIDVALG FRA KOEREGISTER.
ANDNOT C13_IND_VST80_K3  ; Z
SET T04_L3_PAST_IND  ; TIL PASTEURER VIA LINJE 3
LD TR0
AND T05_L3_VALG  ; INDIVIDVALG FRA KOEREGISTER.
ANDNOT C14_IND_VST80_K3  ; Z
SET T05_L3_PAST_IND  ; TIL PASTEURER VIA LINJE 3
; rung 15: INDIVID-RESET
LDNOT SILO_L3_PAST_START  ; program starter
RSET T03_L3_PAST_IND  ; TIL PASTEURER VIA LINJE 3
RSET T04_L3_PAST_IND  ; TIL PASTEURER VIA LINJE 3
RSET T05_L3_PAST_IND  ; TIL PASTEURER VIA LINJE 3
; rung 16: INDIVID-INNE INDIVID ER VALGT
LDNOT T03_L3_PAST_IND  ; TIL PASTEURER VIA LINJE 3
ANDNOT T04_L3_PAST_IND  ; TIL PASTEURER VIA LINJE 3
ANDNOT T05_L3_PAST_IND  ; TIL PASTEURER VIA LINJE 3
OUTNOT SILO_L3_PAST_INDIVID_INNE  ; Individadresse er

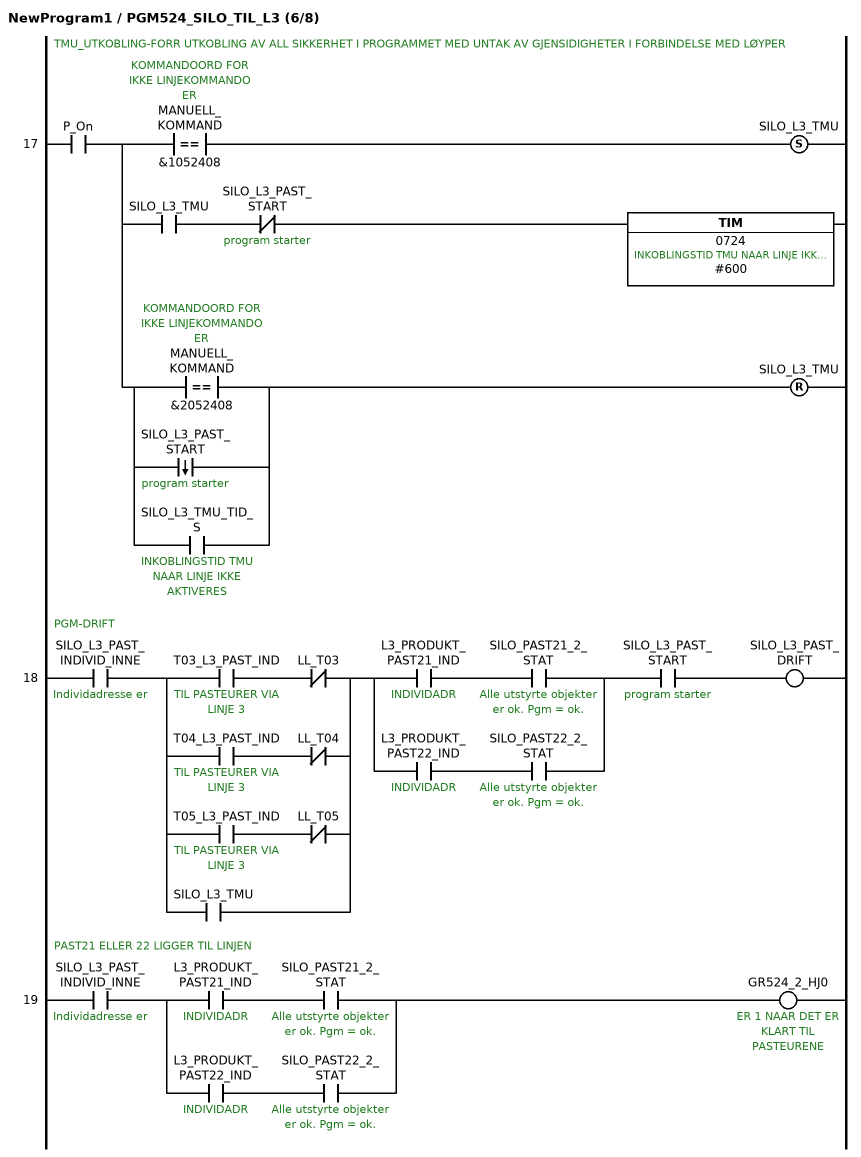
; rung 17: TMU_UTKOBLING-FORR UTKOBLING AV ALL SIKKERHET I PROGRAMMET MED UNTAK AV GJENSIDIGHETER I FORBINDELSE MED LØYPER
LD P_On
OUT TR0
AND=L(301) MANUELL_KOMMAND &1052408  ; KOMMANDOORD FOR IKKE LINJEKOMMANDOER
SET SILO_L3_TMU
LD TR0
AND SILO_L3_TMU
ANDNOT SILO_L3_PAST_START  ; program starter
TIM 0724 #600  ; INKOBLINGSTID TMU NAAR LINJE IKKE AKTIVERES
LD TR0
LD=L(301) MANUELL_KOMMAND &2052408  ; KOMMANDOORD FOR IKKE LINJEKOMMANDOER
%OR SILO_L3_PAST_START  ; program starter
OR SILO_L3_TMU_TID_S  ; INKOBLINGSTID TMU NAAR LINJE IKKE AKTIVERES
ANDLD
RSET SILO_L3_TMU
; rung 18: PGM-DRIFT
LD SILO_L3_PAST_INDIVID_INNE  ; Individadresse er
LD T03_L3_PAST_IND  ; TIL PASTEURER VIA LINJE 3
ANDNOT LL_T03
LD T04_L3_PAST_IND  ; TIL PASTEURER VIA LINJE 3
ANDNOT LL_T04
ORLD
LD T05_L3_PAST_IND  ; TIL PASTEURER VIA LINJE 3
ANDNOT LL_T05
ORLD
OR SILO_L3_TMU
ANDLD
LD L3_PRODUKT_PAST21_IND  ; INDIVIDADR
AND SILO_PAST21_2_STAT  ; Alle utstyrte objekter er ok. Pgm = ok.
LD L3_PRODUKT_PAST22_IND  ; INDIVIDADR
AND SILO_PAST22_2_STAT  ; Alle utstyrte objekter er ok. Pgm = ok.
ORLD
ANDLD
AND SILO_L3_PAST_START  ; program starter
OUT SILO_L3_PAST_DRIFT
; rung 19: PAST21 ELLER 22 LIGGER TIL LINJEN
LD SILO_L3_PAST_INDIVID_INNE  ; Individadresse er
LD L3_PRODUKT_PAST21_IND  ; INDIVIDADR
AND SILO_PAST21_2_STAT  ; Alle utstyrte objekter er ok. Pgm = ok.
LD L3_PRODUKT_PAST22_IND  ; INDIVIDADR
AND SILO_PAST22_2_STAT  ; Alle utstyrte objekter er ok. Pgm = ok.
ORLD
ANDLD
OUT GR524_2_HJ0  ; ER 1 NAAR DET ER KLART TIL PASTEURENE

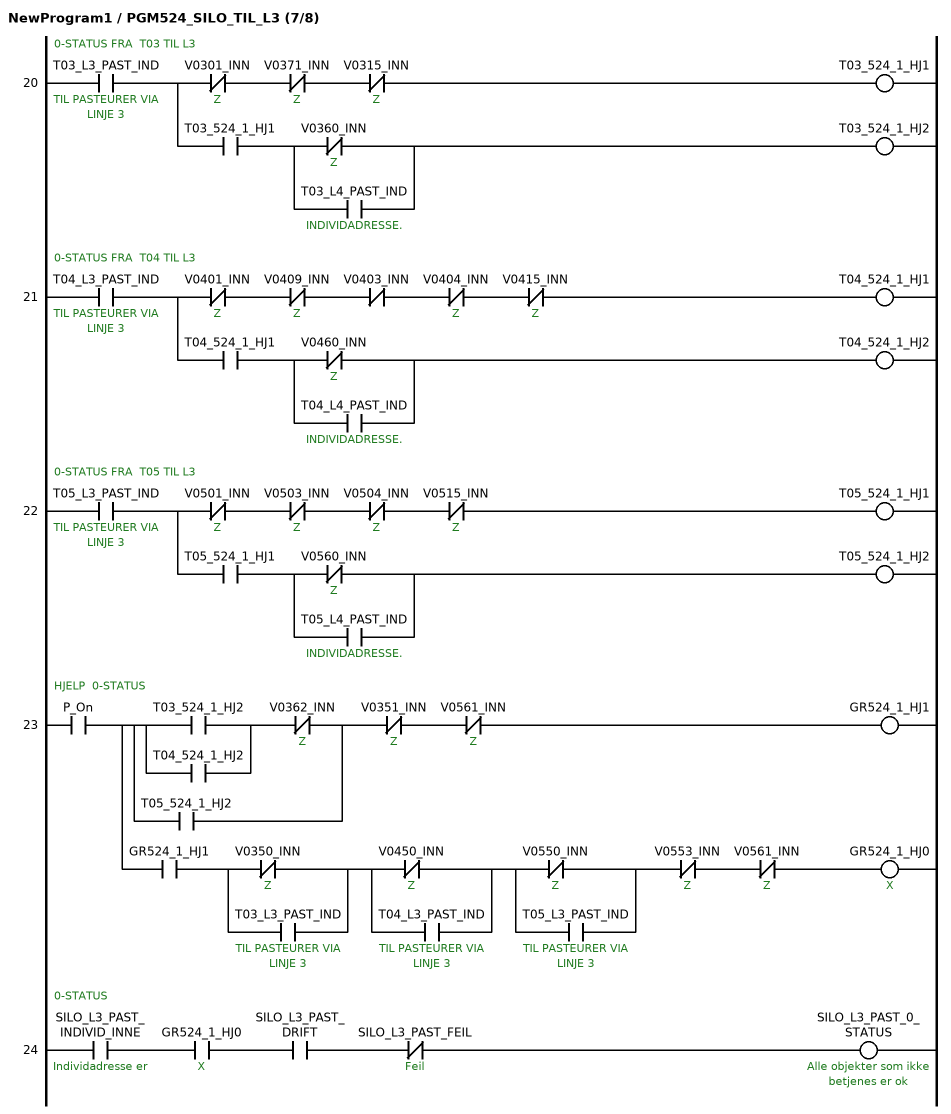
; rung 20: 0-STATUS FRA  T03 TIL L3
LD T03_L3_PAST_IND  ; TIL PASTEURER VIA LINJE 3
OUT TR0
ANDNOT V0301_INN  ; Z
ANDNOT V0371_INN  ; Z
ANDNOT V0315_INN  ; Z
OUT T03_524_1_HJ1
LD TR0
AND T03_524_1_HJ1
LDNOT V0360_INN  ; Z
OR T03_L4_PAST_IND  ; INDIVIDADRESSE.
ANDLD
OUT T03_524_1_HJ2
; rung 21: 0-STATUS FRA  T04 TIL L3
LD T04_L3_PAST_IND  ; TIL PASTEURER VIA LINJE 3
OUT TR0
ANDNOT V0401_INN  ; Z
ANDNOT V0409_INN  ; Z
ANDNOT V0403_INN
ANDNOT V0404_INN  ; Z
ANDNOT V0415_INN  ; Z
OUT T04_524_1_HJ1
LD TR0
AND T04_524_1_HJ1
LDNOT V0460_INN  ; Z
OR T04_L4_PAST_IND  ; INDIVIDADRESSE.
ANDLD
OUT T04_524_1_HJ2
; rung 22: 0-STATUS FRA  T05 TIL L3
LD T05_L3_PAST_IND  ; TIL PASTEURER VIA LINJE 3
OUT TR0
ANDNOT V0501_INN  ; Z
ANDNOT V0503_INN  ; Z
ANDNOT V0504_INN  ; Z
ANDNOT V0515_INN  ; Z
OUT T05_524_1_HJ1
LD TR0
AND T05_524_1_HJ1
LDNOT V0560_INN  ; Z
OR T05_L4_PAST_IND  ; INDIVIDADRESSE.
ANDLD
OUT T05_524_1_HJ2
; rung 23: HJELP  0-STATUS
LD P_On
OUT TR0
LD T03_524_1_HJ2
OR T04_524_1_HJ2
ANDNOT V0362_INN  ; Z
OR T05_524_1_HJ2
ANDLD
ANDNOT V0351_INN  ; Z
ANDNOT V0561_INN  ; Z
OUT GR524_1_HJ1
LD TR0
AND GR524_1_HJ1
LDNOT V0350_INN  ; Z
OR T03_L3_PAST_IND  ; TIL PASTEURER VIA LINJE 3
ANDLD
LDNOT V0450_INN  ; Z
OR T04_L3_PAST_IND  ; TIL PASTEURER VIA LINJE 3
ANDLD
LDNOT V0550_INN  ; Z
OR T05_L3_PAST_IND  ; TIL PASTEURER VIA LINJE 3
ANDLD
ANDNOT V0553_INN  ; Z
ANDNOT V0561_INN  ; Z
OUT GR524_1_HJ0  ; X
; rung 24: 0-STATUS
LD SILO_L3_PAST_INDIVID_INNE  ; Individadresse er
AND GR524_1_HJ0  ; X
AND SILO_L3_PAST_DRIFT
ANDNOT SILO_L3_PAST_FEIL  ; Feil
OUT SILO_L3_PAST_0_STATUS  ; Alle objekter som ikke betjenes er ok

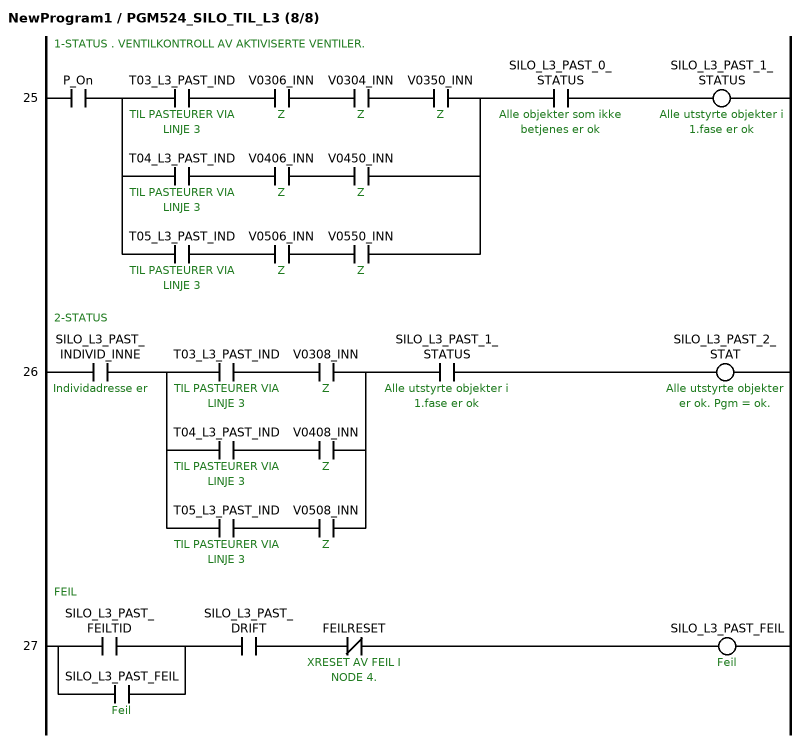
; rung 25: 1-STATUS . VENTILKONTROLL AV AKTIVISERTE VENTILER.
LD P_On
LD T03_L3_PAST_IND  ; TIL PASTEURER VIA LINJE 3
AND V0306_INN  ; Z
AND V0304_INN  ; Z
AND V0350_INN  ; Z
LD T04_L3_PAST_IND  ; TIL PASTEURER VIA LINJE 3
AND V0406_INN  ; Z
AND V0450_INN  ; Z
ORLD
LD T05_L3_PAST_IND  ; TIL PASTEURER VIA LINJE 3
AND V0506_INN  ; Z
AND V0550_INN  ; Z
ORLD
ANDLD
AND SILO_L3_PAST_0_STATUS  ; Alle objekter som ikke betjenes er ok
OUT SILO_L3_PAST_1_STATUS  ; Alle utstyrte objekter i 1.fase er ok
; rung 26: 2-STATUS
LD SILO_L3_PAST_INDIVID_INNE  ; Individadresse er
LD T03_L3_PAST_IND  ; TIL PASTEURER VIA LINJE 3
AND V0308_INN  ; Z
LD T04_L3_PAST_IND  ; TIL PASTEURER VIA LINJE 3
AND V0408_INN  ; Z
ORLD
LD T05_L3_PAST_IND  ; TIL PASTEURER VIA LINJE 3
AND V0508_INN  ; Z
ORLD
ANDLD
AND SILO_L3_PAST_1_STATUS  ; Alle utstyrte objekter i 1.fase er ok
OUT SILO_L3_PAST_2_STAT  ; Alle utstyrte objekter er ok. Pgm = ok.
; rung 27: FEIL
LD SILO_L3_PAST_FEILTID
OR SILO_L3_PAST_FEIL  ; Feil
AND SILO_L3_PAST_DRIFT
ANDNOT FEILRESET  ; XRESET AV FEIL I NODE 4.
OUT SILO_L3_PAST_FEIL  ; Feil

### Section PGM525_SILO_TIL_L4

